Staubli VAL3: deleteItem.pgx

program deleteItem(bool& x_bResult)
  local string l_sMessage
  local string l_sButton[2]
  local string l_sTitle
  local bool l_bYes
begin
  x_bResult=false
  //delete it
  call language2:message(l_sMessage,3)
  call language:getYesNo(l_sButton)
  call set:getListTitle(l_sTitle)
  call use:yes_no(l_sMessage+"#"+l_sTitle+" "+sEvent,l_sButton,l_bYes)
  x_bResult=l_bYes
end
